TYPE TcoDatamanResultData_v_5_x_x : STRUCT
    ResultID AT %I* : UINT;
    ResultCode AT %I* : UINT;
    ResultExtended AT %I* : UINT;
    ResultLength AT %I* : UINT;
    ResultData AT %I* : ARRAY[0..245] OF BYTE;
END_STRUCT
END_TYPE

(* stored: Version 1.1.0.1, ProductVersion 3.1.4024.11
   DUT TcoDatamanResultData_v_5_x_x: Id {f7879786-b132-47dc-823e-6e5cb4dcf1f1} *)
